INTERFACE ITF_SPM_OLD_HMI_Init EXTENDS B_Baza.ITF_Komponent, ITF_SPM_OLD_HMI_Lacznik

END_INTERFACE

(* stored: Version 1.1.0.1
   Itf ITF_SPM_OLD_HMI_Init: Id {9a2e5680-ab26-0a5b-12b8-3d93cda48364} *)
